RoboDK station: jugar_bolos.rdk

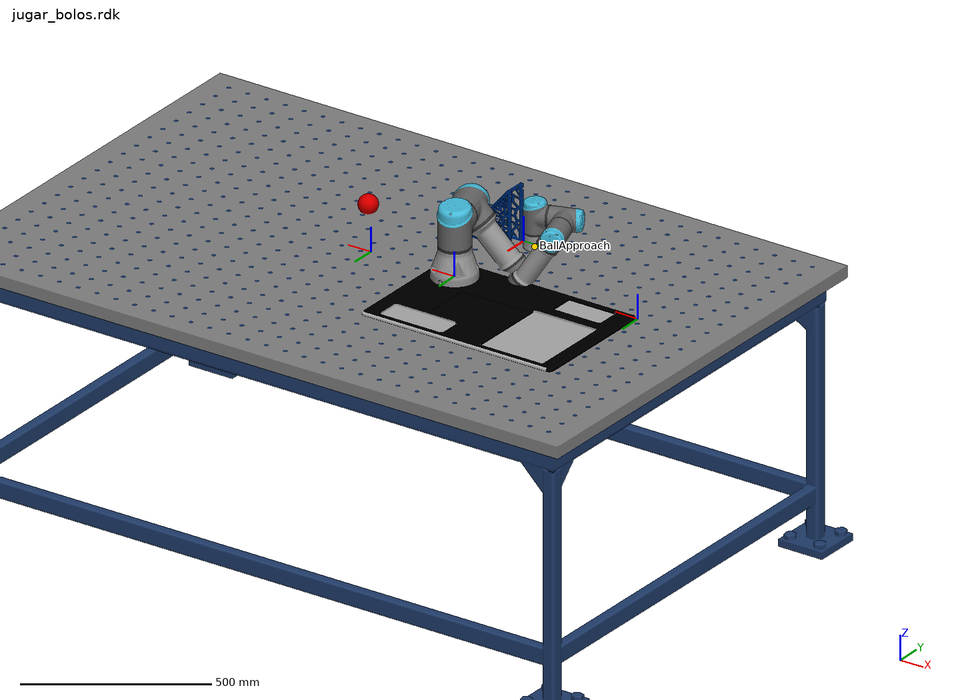
[picture v0: the station drawn from its stored meshes, robots at their saved joint values, targets as dots, program paths as lines]
Station jugar_bolos (saved by RoboDK 5.9.0). Poses are relative to the parent item; angles as X-Y-Z fixed-axis rotations.
  - object Table 2000x1200x800mm at (0, 0, 0) mm, size 2020 x 1340 x 800 mm, geometry from Table-2000x1200x800mm.sld
  - frame rampa at (860, 285, 5) mm, rotated rx 0 ry 0 rz -90 deg
    - object Braquet at (-3, -40, 8) mm, rotated rx 180 ry 0 rz 90 deg, size 5 x 66 x 7 mm, geometry from Braquet.stl
    - object Brazo_D at (60, 0, 0) mm, size 5 x 150 x 168 mm, geometry from Brazo_D.stl
    - object Brazo_I at (0, 0, 0) mm, size 5 x 150 x 168 mm, geometry from Brazo_I.stl
    - object rampa at (60, -150, 0) mm, rotated rx -50 ry 0 rz 180 deg, size 60 x 215.8 x 4 mm, geometry from rampa.stl
  - frame Bola Base at (570, 5, 5) mm, rotated rx 0 ry 0 rz 180 deg
    - robot Bola: 3 axes
        modified DH rows (alpha deg, a mm, theta deg, d mm): 0, 0, 0, 0 linear; 90, 0, 90, 0 linear; 90, 0, 0, 0 linear
        base shift (0, 0, 0) mm, rotated rx 0 ry -90 rz 180 deg
        joint limits [-999999, -999999, -999999] to [999999, 999999, 999999]; home [0, 0, 0]; saved at [136.9, -182, 0]
      - tool 10491_Bowling Ball_v1_max8_iteration-2, TCP at (0, 0, 200) mm, size 54.9 x 54.8 x 55 mm, geometry from 10491_Bowling Ball_v1_max8_iteration-2.obj
  - frame UR3e Base at (840, 0, 10) mm, rotated rx 0 ry 0 rz 180 deg
    - robot UR3e: 6 axes, payload 3 kg, reach 500 mm, repeatability 0.03 mm, weight 11 kg
        modified DH rows (alpha deg, a mm, theta deg, d mm): 0, 0, 0, 151.9; 90, 0, 180, 0; 0, 243.55, 0, 0; 0, 213.2, 0, 131.05; -90, 0, 0, 85.35; 90, 0, 180, 92.1
        joint limits [-360, -360, -360, -360, -360, -360] to [360, 360, 360, 360, 360, 360]; home [0, -90, -90, 0, 90, 0]; saved at [18.787, 51.414, -109.3, 147.885, 90, 108.787]
    - frame BaseRobotUR3e Base at (-525, -85, -10) mm
      - object BaseRobotUR3e at (0, 0, 0) mm, size 610 x 398 x 10 mm, geometry from BaseRobotUR3e.STL
    - target BallApproach (Cartesian target) at (-128.1, -182, 50) mm, rotated rx 180 ry 0 rz 180 deg; joints [-88.694, -231.312, -250.94, 32.252, -90, 181.306] of UR3e
